(* IEC 61131-3 sources: Industry-PLC-LLM/data/PLCBEAD_repo/PLCBEAD_PLCEmbed-main/PLC-BEAD/Source/GEB/MAX3, 1 file *)

(* ---- MAX3.ST ---- *)
FUNCTION MAX3:REAL

	VAR_INPUT
		IN1 :	REAL;
		IN2 :	REAL;
		IN3 :	REAL;
	END_VAR

	MAX3 := MAX(MAX(IN1,IN2),IN3);

END_FUNCTION

PROGRAM program0
	VAR
		IN1 :	REAL;
		IN2 :	REAL;
		IN3 :	REAL;

		OUT : REAL;
	END_VAR

	OUT := MAX3(IN1, IN2, IN3);

END_PROGRAM
